FUNCTION_BLOCK Motor_Conveyor_1 IMPLEMENTS i_Motor
VAR_INPUT
END_VAR
VAR_OUTPUT
END_VAR
VAR
END_VAR

{warning 'add method implementation '}
METHOD Motor_Off : BOOL
END_METHOD

{warning 'add method implementation '}
METHOD Motor_On : BOOL
END_METHOD

END_FUNCTION_BLOCK

(* stored: Version 1.1.0.1, ProductVersion 3.1.4024.11
   POU Motor_Conveyor_1: Id {007fbfa0-f3aa-4518-bc68-198fbeeca44e}, SpecialFunc None
   Method Motor_Off: Id {de3d80f9-e893-4f0f-9369-891afdb69e0b}
   Method Motor_On: Id {0ca6c61e-e247-4933-9cff-197f27f74695} *)
